PROGRAM MAIN
VAR
	
	inner_arm : FB_CalculateLinkageArm; // for HMI and Scope
	outer_arm : FB_CalculateLinkageArm; // for HMI and Scope
	third_arm : FB_CalculateLinkageArm; // for Scope
	z0: REAL := 0; // for 3d scope chart
	
	io_X:	AXIS_REF;
	io_Y:	AXIS_REF;
	io_Z:	AXIS_REF;
	io_C:	AXIS_REF;	
	io_M1:	AXIS_REF;
	io_M2:	AXIS_REF;
	io_M3:	AXIS_REF;
	io_M4:	AXIS_REF;	

	fbAddAxisXtoGrp : MC_AddAxisToGroup;
	fbAddAxisYtoGrp : MC_AddAxisToGroup;
	fbAddAxisZtoGrp : MC_AddAxisToGroup;	
	fbAddAxisCtoGrp : MC_AddAxisToGroup;	
	
//	Kinematic Functions / Structures / Vars
	bkinConfigGrp				: BOOL;
	bkinCartesianMode			: BOOL := TRUE; //When bCartesianMode is TRUE, movement in the MCS (Cartesian) axes will be transformed into the ACS (Joint) axes. The ACS axes cannot be moved directly.
	bkinResetGrp					: BOOL;
	in_stKinToPlc	AT %I*		: NcToPlc_NciChannel_Ref;
	out_stPlcToKin	AT %Q*		: PLCTONC_NCICHANNEL_REF;
	stAxesConfig				: ST_KinAxes;
	fbCalcTrafo					: FB_KinCalcTrafo;
	metaIn						: U_KinMetaInfo;
	metaOut						: U_KinMetaInfo;
	fbKinConfigGrp				: FB_KinConfigGroup;  //Configures ACS and MCS axes to the kinematic transformation group
	fbKinResetGrp				: FB_KinResetGroup;  //Resets the kinematic transformation group
	oidTrafo		AT %I*		: OTCID;
	kinStatus 					: E_KinStatus;
	
	bDeltaKinEnable : BOOL;
	bDeltaKinReady : BOOL;
	bDeltaKinActive : BOOL;
	bDeltaKinInactive : BOOL;
	nDeltaKinState : INT;
	
	bKinGrpEnable : BOOL;
	bKinGrpReady : BOOL;
	bKinGrpError : BOOL;
	bKinGrpReset : BOOL;
	bNciEnable : BOOL;
	bKinResetDone : BOOL;
	bNciReadytToEnable : BOOL;
	bEnableAxes : BOOL;
	bAllAxesReady : BOOL;
	fbKinDelay : TON;
	fbEnableAxes : FB_EnableAxes;
	bAxisFault : BOOL;
	fbResetCoordinateAxes : FB_ResetCoordinateAxes;
	fbJogX : MC_Jog;
	fbJogY : MC_Jog;
	fbJogZ : MC_Jog;
	fbMoveX : MC_MoveRelative;
	bMoveX : BOOL;
	nDistanceX : INT;
	nDistanceY : INT;
	nDistanceZ : INT;
	bMoveY : BOOL;
	bMoveZ : BOOL;
	fbMoveY : MC_MoveRelative;
	fbMoveZ : MC_MoveRelative;
	bAxesNotMoving : BOOL;
	bJogXpos : BOOL;
	bJogXneg : BOOL;
	nMoveState	: WORD;
	
	bMotionGrpEnable : BOOL;	// Enable the Motion Group
	bMotionGrpBuild : BOOL;		// Add Axes To Motion Group
	bMotionGrpStop : BOOL;
	bMotionGrpStart : BOOL;
	bMotionGrpPrep : BOOL;
	bMotionGrpOvr : BOOL;
	
	fbMgSetOverride : MC_GroupSetOverride;
	fbMgEnable : MC_GroupEnable;
	fbMoveLinPrep : MC_MoveLinearAbsolutePreparation;
	fbMoveCircPrep : MC_MoveCircularAbsolutePreparation;
	fbMgMovePath : MC_MovePath;
	fbMgStop 	: MC_GroupStop;
	fbMgReadStatus : MC_GroupReadStatus;
	
	// hmi
	
	nDisplayZ : LREAL;
	nPkgZ   : LREAL;
	nScaleZ : LREAL;
	nDisplayX : LREAL;
	nDisplayY : LREAL;
	
	
	// copied from sample proj
	
	buffer					: ARRAY[1..4096] OF BYTE;
	path					: MC_PATH_DATA_REF(ADR(buffer), SIZEOF(buffer));
	
	aTargetPos				: ARRAY[1..4] OF MC_LREAL;
	aTransitionParam		: ARRAY[1..2] OF MC_LREAL;
	aAuxPoint                               : ARRAY[1..3] OF MC_LREAL;
	fVelFactor				: LREAL := 1.0;
	bMovePrepError : BOOL;
	bBarPicked : BOOL;
	bAddNewBar : BOOL;
	fbAddNewBar : TON;
	bBarPlaced : BOOL;
	nBarDisplayX : LREAL;
	nBarDisplayY : LREAL;
	nBarDisplayZ : LREAL;
	bNewPath	: BOOL;
	bBarInPlace  : BOOL;
	nTestBarX : LREAL;
	nTestBarY : LREAL;
	nTestBarZ : LREAL;
		nScaledBarX : LREAL;
	nScaledBarY : LREAL;
	nScaledBarZ : LREAL;
	
	
	fbTrackConveyor : MC_TrackConveyorBelt;
	MasterRefPos : MC_LREAL;
	InitialObjectPos : ARRAY [1..4] OF MC_LREAL;
	bStartTracking : BOOL;
	fbStartConveyor : MC_MoveVelocity;
	fbStopConveyor : MC_Stop;
	bStartConveyor : BOOL;
	bStopGroup : BOOL;
	lrYpos: MC_LREAL;
	fbSetM1Pos : MC_SetPosition;
	fbSetM2Pos : MC_SetPosition;
	fbSetM4Pos : MC_SetPosition;
	bSetPos : BOOL;
	
	nTrackX: LREAL;
END_VAR


// action calls
	Main.cartesian_ops();
	Main.kinematic_ops();
	Main.motion_group();

// calculations for hmi display of the scara linkages
	inner_arm(
		x0:= 375, 
		y0:= 375, 
		theta:= io_M1.NcToPlc.ActPos, 
		L:= 190, 
		x1=> , 
		y1=> );
	
	outer_arm(
		x0:= inner_arm.x1, 
		y0:= inner_arm.y1, 
		theta:= io_M2.NcToPlc.ActPos, 
		L:= 190, 
		x1=> , 
		y1=> );
	third_arm(
		x0:= outer_arm.x1, 
		y0:= outer_arm.y1, 
		theta:= io_M4.NcToPlc.ActPos, 
		L:= 75, 
		x1=> , 
		y1=> );
	z0;
	

// Axis Ref Read Status
	io_X.ReadStatus();
	io_Y.ReadStatus();
	io_Z.ReadStatus();
	io_C.ReadStatus();	
	io_M1.ReadStatus();
	io_M2.ReadStatus();
	io_M3.ReadStatus();
	io_M4.ReadStatus();	

// check for motor movement
	bAxesNotMoving := io_M1.Status.NotMoving AND io_M2.Status.NotMoving AND io_M3.Status.NotMoving AND io_M4.Status.NotMoving;
	
// read axes id's from cylic interface so they can mapped later to the kinematic group
	stAxesConfig.nAxisIdsAcs[1]	:= io_M1.NcToPlc.AxisId;
	stAxesConfig.nAxisIdsAcs[2]	:= io_M2.NcToPlc.AxisId;
	stAxesConfig.nAxisIdsAcs[3]	:= io_M3.NcToPlc.AxisId;
	stAxesConfig.nAxisIdsAcs[4]	:= io_M4.NcToPlc.AxisId;	
	stAxesConfig.nAxisIdsMcs[1]	:= io_X.NcToPlc.AxisId;
	stAxesConfig.nAxisIdsMcs[2]	:= io_Y.NcToPlc.AxisId;
	stAxesConfig.nAxisIdsMcs[3]	:= io_Z.NcToPlc.AxisId;
	stAxesConfig.nAxisIdsMcs[4]	:= io_C.NcToPlc.AxisId;	
	

	fbMgMovePath(
		AxesGroup:= GVL.stGroupRef , 
		PathData:= path , 
		Execute:= bMotionGrpStart
	);
	
	fbMgStop(
		AxesGroup := GVL.stGroupRef,
		Execute	:= bStopGroup
		);
	
			
CASE nMoveState OF
	
1:	//	init

		nMoveState	:= 4;
		
4:	// set up path data for the pick position

		Main.prep_pick_path();
		//Main.prep_start_path();
		
		IF path.FilledRows > 0 THEN
			nMoveState	:= 5;
		END_IF
		
5:	// move to the pick psoition

		bMotionGrpStart := TRUE;

		IF fbMgMovePath.Done THEN
			bMotionGrpStart := FALSE;
			nMoveState := 100;
		END_IF

10:	// set up path data for the place position

		Main.prep_place_path();
		//Main.prep_finish_path();
		
		IF path.FilledRows > 0 THEN
			nMoveState	:= 15;
		END_IF
		
15:	// move to the place position

		bMotionGrpStart := TRUE;

		IF fbMgMovePath.Done THEN
			bMotionGrpStart := FALSE;
			nMoveState := 1;
		END_IF

100: // stopping...

		bStopGroup := TRUE;
		
		IF fbMgStop.Done THEN
			bStopGroup := FALSE;
			nMoveState	:= 10;
		END_IF		

END_CASE

ACTION cartesian_ops:
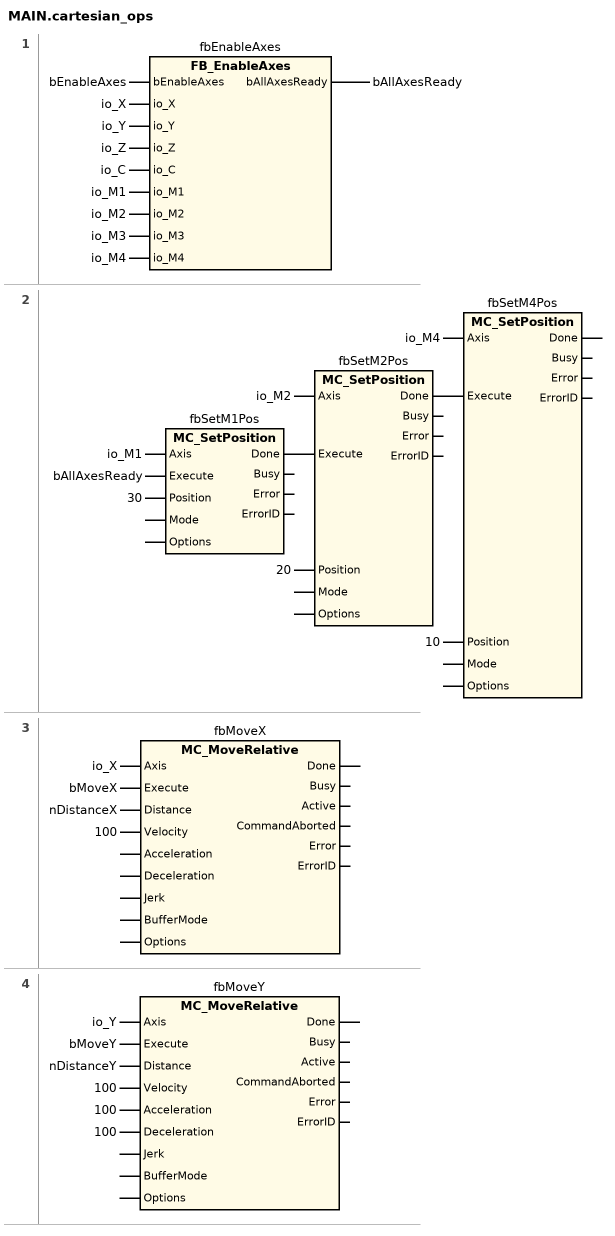
// NETWORK 1
fbEnableAxes(
    bEnableAxes := bEnableAxes,
    io_X := io_X,
    io_Y := io_Y,
    io_Z := io_Z,
    io_C := io_C,
    io_M1 := io_M1,
    io_M2 := io_M2,
    io_M3 := io_M3,
    io_M4 := io_M4); // FB_EnableAxes
bAllAxesReady := fbEnableAxes.bAllAxesReady;

// NETWORK 2
fbSetM1Pos(Axis := io_M1, Execute := bAllAxesReady, Position := 30); // MC_SetPosition
fbSetM2Pos(Axis := io_M2, Execute := fbSetM1Pos.Done, Position := 20); // MC_SetPosition
fbSetM4Pos(Axis := io_M4, Execute := fbSetM2Pos.Done, Position := 10); // MC_SetPosition

// NETWORK 3
fbMoveX(Axis := io_X, Execute := bMoveX, Distance := nDistanceX, Velocity := 100); // MC_MoveRelative

// NETWORK 4
fbMoveY(
    Axis := io_Y,
    Execute := bMoveY,
    Distance := nDistanceY,
    Velocity := 100,
    Acceleration := 100,
    Deceleration := 100); // MC_MoveRelative

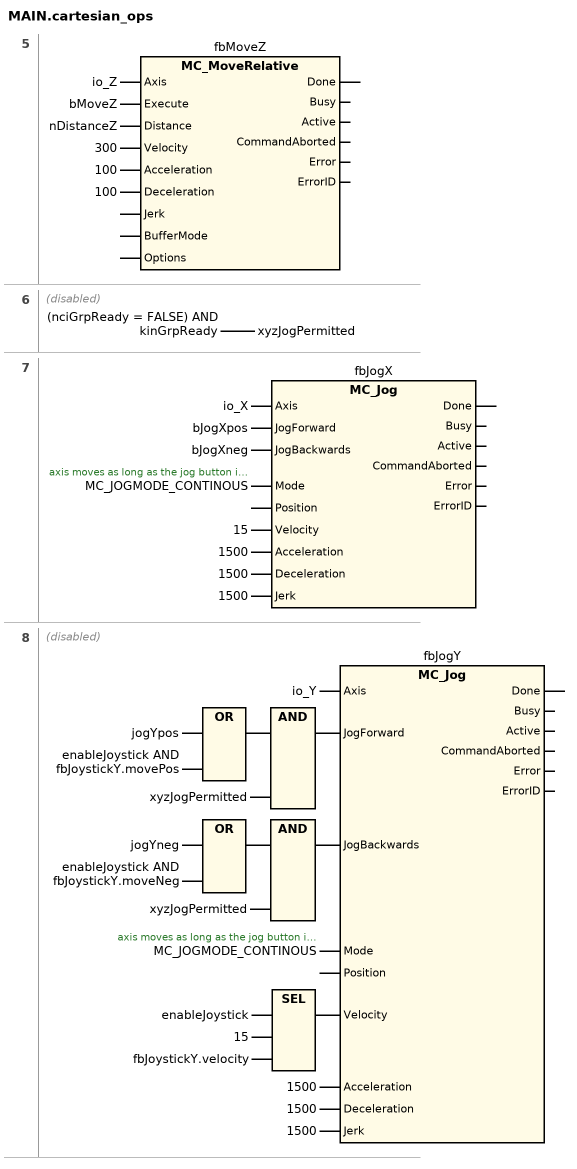
// NETWORK 5
fbMoveZ(
    Axis := io_Z,
    Execute := bMoveZ,
    Distance := nDistanceZ,
    Velocity := 300,
    Acceleration := 100,
    Deceleration := 100); // MC_MoveRelative

// NETWORK 6 (disabled)
// xyzJogPermitted := (nciGrpReady = FALSE) AND kinGrpReady;

// NETWORK 7
//   MC_JOGMODE_CONTINOUS: axis moves as long as the jog button is pressed using parameterized dynamics
fbJogX(
    Axis := io_X,
    JogForward := bJogXpos,
    JogBackwards := bJogXneg,
    Mode := MC_JOGMODE_CONTINOUS,
    Velocity := 15,
    Acceleration := 1500,
    Deceleration := 1500,
    Jerk := 1500); // MC_Jog

// NETWORK 8 (disabled)
//   MC_JOGMODE_CONTINOUS: axis moves as long as the jog button is pressed using parameterized dynamics
// fbJogY(
//     Axis := io_Y,
//     JogForward := (jogYpos OR (enableJoystick AND fbJoystickY.movePos)) AND xyzJogPermitted,
//     JogBackwards := (jogYneg OR (enableJoystick AND fbJoystickY.moveNeg)) AND xyzJogPermitted,
//     Mode := MC_JOGMODE_CONTINOUS,
//     Velocity := SEL(enableJoystick, 15, fbJoystickY.velocity),
//     Acceleration := 1500,
//     Deceleration := 1500,
//     Jerk := 1500); // MC_Jog

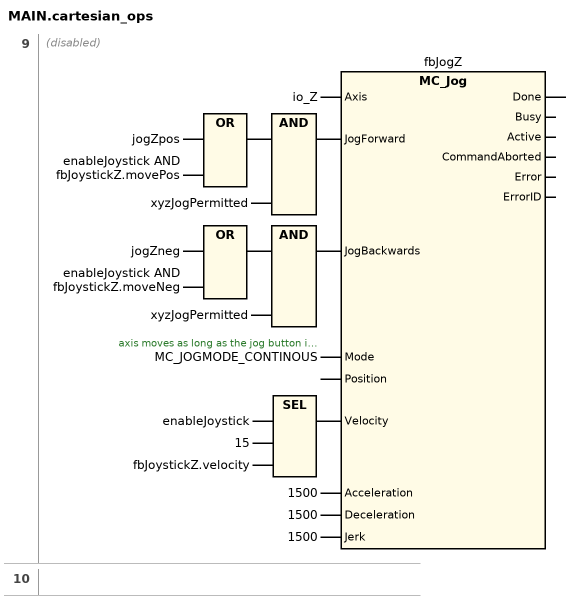
// NETWORK 9 (disabled)
//   MC_JOGMODE_CONTINOUS: axis moves as long as the jog button is pressed using parameterized dynamics
// fbJogZ(
//     Axis := io_Z,
//     JogForward := (jogZpos OR (enableJoystick AND fbJoystickZ.movePos)) AND xyzJogPermitted,
//     JogBackwards := (jogZneg OR (enableJoystick AND fbJoystickZ.moveNeg)) AND xyzJogPermitted,
//     Mode := MC_JOGMODE_CONTINOUS,
//     Velocity := SEL(enableJoystick, 15, fbJoystickZ.velocity),
//     Acceleration := 1500,
//     Deceleration := 1500,
//     Jerk := 1500); // MC_Jog

// NETWORK 10
END_ACTION

ACTION kinematic_ops:
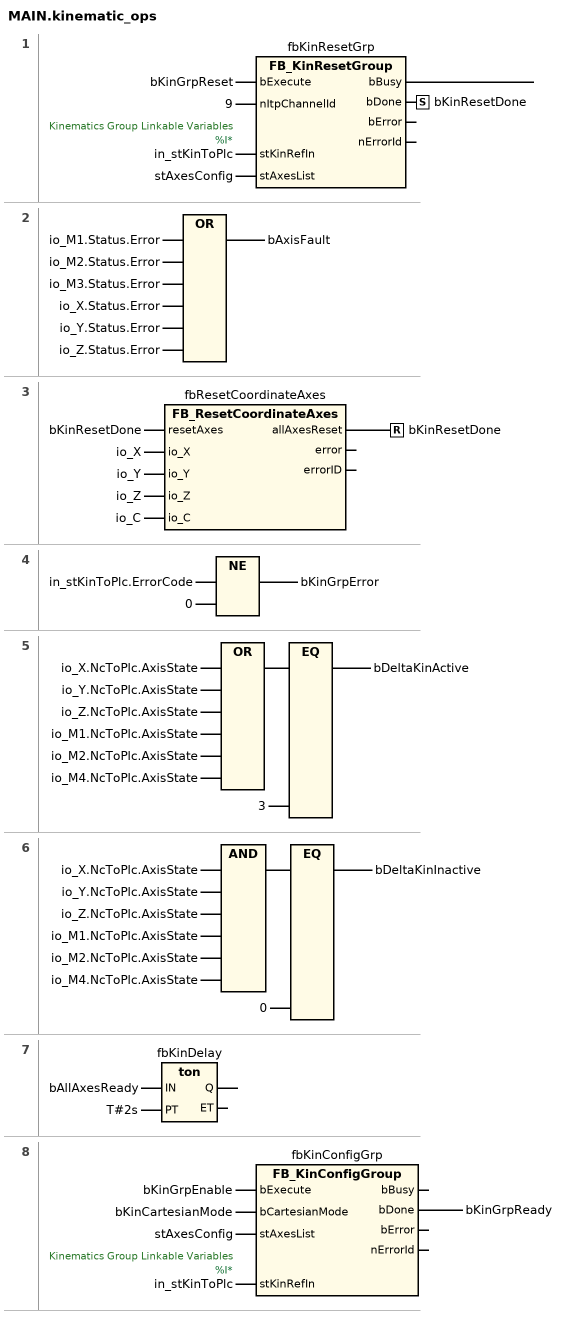
// NETWORK 1
//   fbKinResetGrp: Resets the kinematic transformation group
//   in_stKinToPlc: Kinematics Group Linkable Variables | AT %I*
fbKinResetGrp(
    bExecute := bKinGrpReset,
    nItpChannelId := 9,
    stKinRefIn := in_stKinToPlc,
    stAxesList := stAxesConfig); // FB_KinResetGroup
bKinResetDone S= fbKinResetGrp.bDone;

// NETWORK 2
bAxisFault := io_M1.Status.Error OR io_M2.Status.Error OR io_M3.Status.Error OR io_X.Status.Error OR io_Y.Status.Error OR io_Z.Status.Error;

// NETWORK 3
fbResetCoordinateAxes(resetAxes := bKinResetDone, io_X := io_X, io_Y := io_Y, io_Z := io_Z, io_C := io_C); // FB_ResetCoordinateAxes
bKinResetDone R= fbResetCoordinateAxes.allAxesReset;

// NETWORK 4
bKinGrpError := in_stKinToPlc.ErrorCode <> 0;

// NETWORK 5
bDeltaKinActive := (io_X.NcToPlc.AxisState OR io_Y.NcToPlc.AxisState OR io_Z.NcToPlc.AxisState OR io_M1.NcToPlc.AxisState OR io_M2.NcToPlc.AxisState OR io_M4.NcToPlc.AxisState) = 3;

// NETWORK 6
bDeltaKinInactive := (io_X.NcToPlc.AxisState AND io_Y.NcToPlc.AxisState AND io_Z.NcToPlc.AxisState AND io_M1.NcToPlc.AxisState AND io_M2.NcToPlc.AxisState AND io_M4.NcToPlc.AxisState) = 0;

// NETWORK 7
fbKinDelay(IN := bAllAxesReady, PT := T#2s); // ton

// NETWORK 8
//   fbKinConfigGrp: Configures ACS and MCS axes to the kinematic transformation group
//   in_stKinToPlc: Kinematics Group Linkable Variables | AT %I*
fbKinConfigGrp(
    bExecute := bKinGrpEnable,
    bCartesianMode := bKinCartesianMode,
    stAxesList := stAxesConfig,
    stKinRefIn := in_stKinToPlc); // FB_KinConfigGroup
bKinGrpReady := fbKinConfigGrp.bDone;

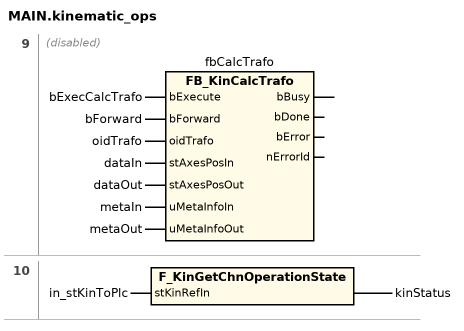
// NETWORK 9 (disabled)
// fbCalcTrafo(
//     bExecute := bExecCalcTrafo,
//     bForward := bForward,
//     oidTrafo := oidTrafo,
//     stAxesPosIn := dataIn,
//     stAxesPosOut := dataOut,
//     uMetaInfoIn := metaIn,
//     uMetaInfoOut := metaOut); // FB_KinCalcTrafo

// NETWORK 10
kinStatus := F_KinGetChnOperationState(stKinRefIn := in_stKinToPlc);
END_ACTION

ACTION kinematic_sm:

(*
		setStartPos[5](Axis:= io_X, 
			Execute:= setZeroPosition,
			Position:= 0);
		setStartPos[6](Axis:= io_Y,
			Execute:= setZeroPosition, 
			Position:= 0);
		setStartPos[7](Axis:= io_Z, 
			Execute:= setZeroPosition,
			Position:= 0);
*)

CASE nDeltaKinState OF 

0: 	nDeltaKinState := 2;

		
2:			// RESET ALL NCI VARIABLES
		//nciRunProgram := FALSE;
		//nciBuildTable := FALSE;
		//nciResetTable := TRUE;
		//nciResetProgram := TRUE;
		nDeltaKinState := 3;
		
3:
		//nciResetProgram := FALSE;
		//nciResetTable := FALSE;
		nDeltaKinState := 4;
		
4:			// RESET ALL KINEMATIC VARIABLES
		IF bKinGrpError THEN
				bKinGrpReset := TRUE;
				nDeltaKinState :=5;
		ELSIF bKinGrpError = FALSE THEN
				nDeltaKinState := 104;
		END_IF
				
5:
		bKinGrpReset := FALSE;
		nDeltaKinState := 4;
		
104:		// RESET ALL KINEMATIC VARIABLES
		IF bAxisFault THEN
				bKinGrpReset := TRUE;
				nDeltaKinState :=105;
		ELSIF bAxisFault = FALSE THEN
				nDeltaKinState := 6;
		END_IF
				
105:
		bKinGrpReset := FALSE;
		nDeltaKinState := 104;

6: 		// IF IN START POSITION - ENABLE AXES
		nDeltaKinState := 7;

7:			// ALL AXES ARE POWERED
		IF bAllAxesReady AND bAxesNotMoving THEN
				nDeltaKinState := 8;
		END_IF
		
8:			// ENABLE KINEMATIC GROUP FUNCTION
		nDeltaKinState := 9;
			
9: 		// DELAY TO ALLOW KINEMATIC GROUP TIME TO PROCESS REQUEST
		IF fbKinDelay.Q AND bKinGrpReady AND bAxesNotMoving THEN
				nDeltaKinState := 10;
		END_IF
	(*	
10:		// ENABLE NCI BUILD GROUP

		nDeltaKinState := 11;

11: 	// WAIT FOR BUILD GROUP DONE AND ADDITIONAL DELAY BEFORE STARTING BUILD TABLE
		IF kinGrpReady  AND  tNciDelay.Q THEN 
				nciBuildTable := TRUE;
				nDeltaKinState := 12;
		ELSIF kinGrpReady = FALSE THEN
				nDeltaKinState := 50;
		END_IF

12: 	// WAIT FOR ROWS TO BE FILLED

		IF fbNciFeedTablePrep.nFilledRows > 0 THEN
				nciBuildTable := FALSE;
				nDeltaKinState:= 13;
		END_IF

13:	// RUN COMMAND WILL START THE NCI FEED TABLE PROGRAM
		IF nciRunCmd  THEN
				nciRunProgram := TRUE; 	
				nDeltaKinState :=14;
		ELSIF nciEnable = FALSE THEN
				nDeltaKinState := 0;
		END_IF
		
14:	
		IF nciFeedingDone THEN
				nciRunProgram := FALSE;
				nDeltaKinState := 15;
		ELSIF nciEnable = FALSE THEN
				nDeltaKinState := 0;
		END_IF

15:	// REACHED END OF FEED TABLE PROGRAM
		IF fbNciTable.bChannelDone THEN
				nDeltaKinState	:= 16;
		ELSIF nciEnable = FALSE THEN
				nDeltaKinState := 0;
		END_IF
		
16:	// IF RUN IS STILL ACTIVE, LOOP BACK THROUGH THE FEED TABLE PROGRAM

		nDeltaKinState := 13;


50: // DECOUPLE KINEMATIC GROUP FROM AXES
		kinCartesianMode := FALSE;
		kinGrpEnable := TRUE;
		
		IF kinStatus = KinStatus_Empty THEN
				kinCartesianMode := TRUE;
				kinGrpEnable := FALSE;
				nDeltaKinState := 4;
		END_IF
	*)			
END_CASE
END_ACTION

ACTION motion_group:
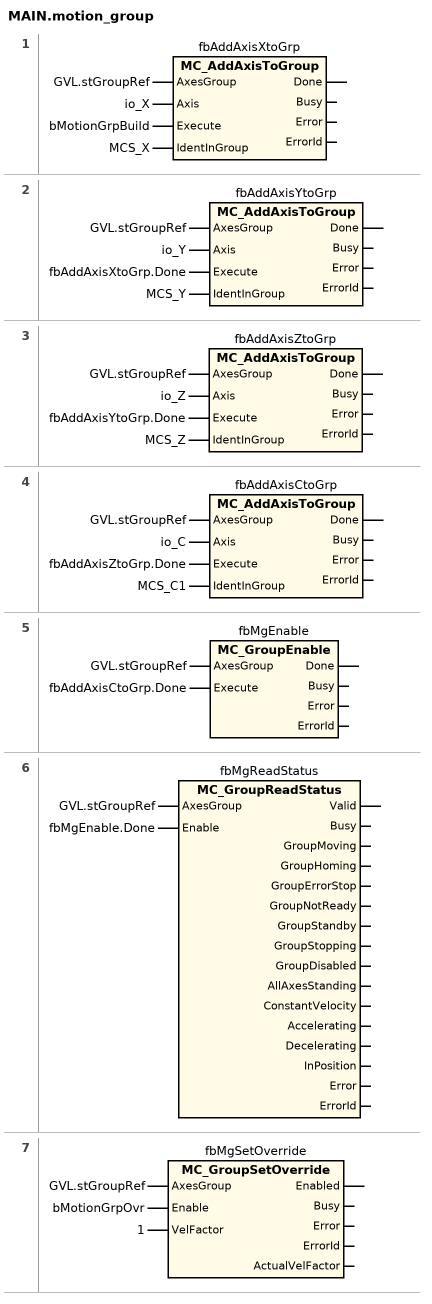
// NETWORK 1
fbAddAxisXtoGrp(AxesGroup := GVL.stGroupRef, Axis := io_X, Execute := bMotionGrpBuild, IdentInGroup := MCS_X); // MC_AddAxisToGroup

// NETWORK 2
fbAddAxisYtoGrp(
    AxesGroup := GVL.stGroupRef,
    Axis := io_Y,
    Execute := fbAddAxisXtoGrp.Done,
    IdentInGroup := MCS_Y); // MC_AddAxisToGroup

// NETWORK 3
fbAddAxisZtoGrp(
    AxesGroup := GVL.stGroupRef,
    Axis := io_Z,
    Execute := fbAddAxisYtoGrp.Done,
    IdentInGroup := MCS_Z); // MC_AddAxisToGroup

// NETWORK 4
fbAddAxisCtoGrp(
    AxesGroup := GVL.stGroupRef,
    Axis := io_C,
    Execute := fbAddAxisZtoGrp.Done,
    IdentInGroup := MCS_C1); // MC_AddAxisToGroup

// NETWORK 5
fbMgEnable(AxesGroup := GVL.stGroupRef, Execute := fbAddAxisCtoGrp.Done); // MC_GroupEnable

// NETWORK 6
fbMgReadStatus(AxesGroup := GVL.stGroupRef, Enable := fbMgEnable.Done); // MC_GroupReadStatus

// NETWORK 7
fbMgSetOverride(AxesGroup := GVL.stGroupRef, Enable := bMotionGrpOvr, VelFactor := 1); // MC_GroupSetOverride
END_ACTION

ACTION prep_finish_path:

path.ClearPath();  //Clear nodes that were in path


// XYZ POSITIONS LIMITS
// X : -760 to +760
// Y : -760 to +760
// Z : 



fbMoveCircPrep.EndPoint                 	:= ADR(aTargetPos);
fbMoveCircPrep.EndPointCount            	:= 4;
fbMoveCircPrep.AuxPoint                 	:= ADR(aTransitionParam);
fbMoveCircPrep.AuxPointCount            	:= 3;
fbMoveCircPrep.CircMode                 	:= mcCircModeCenter;
fbMoveCircPrep.TransitionParameter      	:= ADR(aTransitionParam);
fbMoveCircPrep.TransitionParameterCount 	:= 2;
fbMoveCircPrep.BufferMode               	:= mcBlendingPrevious;
fbMoveCircPrep.TransitionMode           	:= mcTransModeNone;
	
fbMoveLinPrep.Position						:= ADR(aTargetPos); //pointer to position array
fbMoveLinPrep.PositionCount 				:= 4; //number of axes in group
fbMoveLinPrep.TransitionParameter			:= ADR (aTransitionParam); //pointer to transition parameter array
fbMoveLinPrep.TransitionParameterCount		:= 2; //number of transition parameters, has to be set always 2
fbMoveLinPrep.BufferMode					:= mcBlendingPrevious;
fbMoveLinPrep.TransitionMode				:= mcTransModeCornerDistanceAdvanced;

//Set dynamics to default values of the axes
fbMoveLinPrep.Acceleration					:= MC_DEFAULT;
fbMoveLinPrep.Deceleration					:= MC_DEFAULT;
fbMoveLinPrep.Jerk							:= MC_DEFAULT;

bMovePrepError := bMovePrepError OR fbMoveLinPrep.Error;



  	aTargetPos[1]                           := 625;
    aTargetPos[2]                           := 10;
    aTargetPos[3]                           := 0;
    aTransitionParam[1]                     := 0;
    aTransitionParam[2]                     := 0;
    fbMoveLinPrep(PathData:= path, Velocity:= 100, InvokeId:= 10);

    aTargetPos[1]                           := -400;
    aTargetPos[2]                           := -300;
    aTargetPos[3]                           := 0;
    aAuxPoint[1]                            := -357.5;
    aAuxPoint[2]                            := -257.5;
    aAuxPoint[3]                            := 0;
    aTransitionParam[1]                     := 0;
    aTransitionParam[2]                     := 0;
    fbMoveCircPrep(PathData:= path, PathChoice:= mcCircPathchoiceClockwise, Velocity:= 100, InvokeId:= 20);
END_ACTION

ACTION prep_pick_path:
path.ClearPath();  //Clear nodes that were in path


// XYZ POSITIONS LIMITS
// X : -760 to +760
// Y : -760 to +760
// Z : 

//1st node
aTargetPos[1]				:=634;		// X Position
aTargetPos[2]				:= 10;		// Y Position
aTargetPos[3]				:= 0;	// Z Position
aTargetPos[4]				:= 0;	// C Position
aTransitionParam[1]			:= 0; //blending distance on previous segment, no influence here
aTransitionParam[2]			:= 0; //blending distance on this segment, no influence here
fbMoveLinPrep(PathData:= path , Velocity:= 200, InvokeId:= 10);
bMovePrepError := bMovePrepError OR fbMoveLinPrep.Error;

fbMoveLinPrep.Position						:= ADR(aTargetPos); //pointer to position array
fbMoveLinPrep.PositionCount 				:= 4; //number of axes in group
fbMoveLinPrep.TransitionParameter			:= ADR (aTransitionParam); //pointer to transition parameter array
fbMoveLinPrep.TransitionParameterCount		:= 2; //number of transition parameters, has to be set always 2
fbMoveLinPrep.BufferMode					:= mcBlendingPrevious;
fbMoveLinPrep.TransitionMode				:= mcTransModeCornerDistanceAdvanced;
//Set dynamics to default values of the axes
fbMoveLinPrep.Acceleration					:= MC_DEFAULT;
fbMoveLinPrep.Deceleration					:= MC_DEFAULT;
fbMoveLinPrep.Jerk							:= MC_DEFAULT;
END_ACTION

ACTION prep_place_path:
path.ClearPath();  //Clear nodes that were in path

// XYZ POSITIONS LIMITS
// X : -550 to +550
// Y : -550 to +550
// Z : -750 to -950

fbMoveLinPrep.Position						:= ADR(aTargetPos); //pointer to position array
fbMoveLinPrep.PositionCount 				:= 4; //number of axes in group
fbMoveLinPrep.TransitionParameter			:= ADR (aTransitionParam); //pointer to transition parameter array
fbMoveLinPrep.TransitionParameterCount		:= 2; //number of transition parameters, has to be set always 2
fbMoveLinPrep.BufferMode					:= mcBlendingPrevious;
fbMoveLinPrep.TransitionMode				:= mcTransModeCornerDistanceAdvanced;
//Set dynamics to default values of the axes
fbMoveLinPrep.Acceleration					:= MC_DEFAULT;
fbMoveLinPrep.Deceleration					:= MC_DEFAULT;
fbMoveLinPrep.Jerk							:= MC_DEFAULT;
(*
//1st node
aTargetPos[1]				:= -225;		// X Position
aTargetPos[2]				:= 225;		// Y Position
aTargetPos[3]				:= -900;	// Z Position
aTransitionParam[1]			:= 0; //blending distance on previous segment, no influence here
aTransitionParam[2]			:= 0; //blending distance on this segment, no influence here
fbMoveLinPrep(PathData:= path , Velocity:= 2100, InvokeId:= 10);
bMovePrepError := bMovePrepError OR fbMoveLinPrep.Error;

aTargetPos[1]				:= 225;
aTargetPos[2]				:= -225;
aTargetPos[3]				:= -750;
aTransitionParam[1]			:= 50; //blending distance on previous segment (InvokeId=10), defines when to leave line
aTransitionParam[2]			:= 50; //blending distance on this segment, defines latest positionn to be back  on line of InovkeId=20 
fbMoveLinPrep(PathData:= path , Velocity:= 2100, InvokeId:= 20); 
bMovePrepError := bMovePrepError OR fbMoveLinPrep.Error;

aTargetPos[1]				:= 225;
aTargetPos[2]				:= 225;
aTargetPos[3]				:= -950;
aTransitionParam[1]			:= 50; 
aTransitionParam[2]			:= 50;
fbMoveLinPrep(PathData:= path , Velocity:= 2100, InvokeId:= 30);
bMovePrepError := bMovePrepError OR fbMoveLinPrep.Error;

aTargetPos[1]				:= -225;
aTargetPos[2]				:= -225;
aTargetPos[3]				:= -750;
aTransitionParam[1]			:= 50; //blending distance on previous segment, no influence here
aTransitionParam[2]			:= 50; //blending distance on this segment, no influence here
fbMoveLinPrep(PathData:= path , Velocity:= 2100, InvokeId:= 40);
bMovePrepError := bMovePrepError OR fbMoveLinPrep.Error;
*)
aTargetPos[1]				:= -400;
aTargetPos[2]				:= -300;
aTargetPos[3]				:= 0;
aTargetPos[4]				:= 0;
aTransitionParam[1]			:= 50; 
aTransitionParam[2]			:= 50;
fbMoveLinPrep(PathData:= path , Velocity:= 150, InvokeId:= 50);
bMovePrepError := bMovePrepError OR fbMoveLinPrep.Error;
END_ACTION

ACTION prep_start_path:

path.ClearPath();  //Clear nodes that were in path


// XYZ POSITIONS LIMITS
// X : -760 to +760
// Y : -760 to +760
// Z : 



fbMoveCircPrep.EndPoint                 	:= ADR(aTargetPos);
fbMoveCircPrep.EndPointCount            	:= 4;
fbMoveCircPrep.AuxPoint                 	:= ADR(aTransitionParam);
fbMoveCircPrep.AuxPointCount            	:= 3;
fbMoveCircPrep.CircMode                 	:= mcCircModeCenter;
fbMoveCircPrep.TransitionParameter      	:= ADR(aTransitionParam);
fbMoveCircPrep.TransitionParameterCount 	:= 2;
fbMoveCircPrep.BufferMode               	:= mcBlendingPrevious;
fbMoveCircPrep.TransitionMode           	:= mcTransModeNone;
	
fbMoveLinPrep.Position						:= ADR(aTargetPos); //pointer to position array
fbMoveLinPrep.PositionCount 				:= 4; //number of axes in group
fbMoveLinPrep.TransitionParameter			:= ADR (aTransitionParam); //pointer to transition parameter array
fbMoveLinPrep.TransitionParameterCount		:= 2; //number of transition parameters, has to be set always 2
fbMoveLinPrep.BufferMode					:= mcBlendingPrevious;
fbMoveLinPrep.TransitionMode				:= mcTransModeCornerDistanceAdvanced;

//Set dynamics to default values of the axes
fbMoveLinPrep.Acceleration					:= MC_DEFAULT;
fbMoveLinPrep.Deceleration					:= MC_DEFAULT;
fbMoveLinPrep.Jerk							:= MC_DEFAULT;

bMovePrepError := bMovePrepError OR fbMoveLinPrep.Error;



  	aTargetPos[1]                           := -350;
    aTargetPos[2]                           := -300;
    aTargetPos[3]                           := 0;
    aTransitionParam[1]                     := 0;
    aTransitionParam[2]                     := 0;
    fbMoveLinPrep(PathData:= path, Velocity:= 100, InvokeId:= 10);

    aTargetPos[1]                           := 625;
    aTargetPos[2]                           := -10;
    aTargetPos[3]                           := 0;
    aAuxPoint[1]                            := 282.5;
    aAuxPoint[2]                            := -642.5;
    aAuxPoint[3]                            := 0;
    aTransitionParam[1]                     := 0;
    aTransitionParam[2]                     := 0;
    fbMoveCircPrep(PathData:= path, PathChoice:= mcCircPathChoiceCounterClockwise, Velocity:= 100, InvokeId:= 20);
END_ACTION

END_PROGRAM

(* stored: Version 1.1.0.1, ProductVersion 3.1.4024.14
   POU MAIN: Id {fbd90d20-4b58-4f0a-bd6d-ee42c96865f1}, SpecialFunc None
   Action cartesian_ops: Id {b53035e6-9bf1-4fd9-9ba8-c2a72630ca21}
   Action kinematic_ops: Id {c4891f60-7bf3-49b3-b0a9-ddb46ebc1d6c}
   Action kinematic_sm: Id {bbb5d126-a01e-4bc6-9665-181c414ec9e9}
   Action motion_group: Id {dec32b7d-78f0-4b73-bb5d-5b50f024c7db}
   Action prep_finish_path: Id {7e69e7d6-b14f-4a42-9259-a470e72452e9}
   Action prep_pick_path: Id {db426818-fc48-4a7a-861c-8a5631c400aa}
   Action prep_place_path: Id {1209e9dd-a340-4242-82a3-09f8984e11a7}
   Action prep_start_path: Id {9c11d844-023d-493e-a7de-2377b9197ae8} *)
